TYPE Print_Inputs_typ:
STRUCT
	PrintActive AT %I*: BOOL;
	PrintComplete AT %I*: BOOL;
END_STRUCT
END_TYPE

(* stored: Version 1.1.0.1, ProductVersion 3.1.4024.12
   DUT Print_Inputs_typ: Id {71e93a11-43e7-0666-307d-a7a8df27bec1} *)
